# B&R Automation Studio project BuildServer
Automation Studio 4.12.5.95 SP

## Configuration Simulator

CPU PC_any, AutomationRuntime J4.93, Build 4.1.2, Vc V4.72.6

### Hardware
```
PC : PC_any v1.1.1.0 (OrderNumber=PC)
```

## Logical view

### Program Logical/Program

#### Variables.var
```iecst
VAR
	test : UDINT;
	test2 : UDINT;
END_VAR
```

#### Main.st
```iecst
PROGRAM _INIT
	(* Insert code here *)

END_PROGRAM

PROGRAM _CYCLIC
	(* Insert code here *)
	 test := test + 1;
	 test2 := test2 + 1;
END_PROGRAM

PROGRAM _EXIT
	(* Insert code here *)

END_PROGRAM
```
